(* ===== OUTER 10 ===== *)
GVL_test.stCase.aOuters[10].sOuterCode    := 'OUTER10';
GVL_test.stCase.aOuters[10].nOutersStatus := 5;
// packs 1..10
GVL_test.stCase.aOuters[10].aPacks[1].sPackCode   := 'PACK01OUTER10';
GVL_test.stCase.aOuters[10].aPacks[1].nPackStatus := 5;
GVL_test.stCase.aOuters[10].aPacks[2].sPackCode   := 'PACK02OUTER10';
GVL_test.stCase.aOuters[10].aPacks[2].nPackStatus := 5;
GVL_test.stCase.aOuters[10].aPacks[3].sPackCode   := 'PACK03OUTER10';
GVL_test.stCase.aOuters[10].aPacks[3].nPackStatus := 5;
GVL_test.stCase.aOuters[10].aPacks[4].sPackCode   := 'PACK04OUTER10';
GVL_test.stCase.aOuters[10].aPacks[4].nPackStatus := 5;
GVL_test.stCase.aOuters[10].aPacks[5].sPackCode   := 'PACK05OUTER10';
GVL_test.stCase.aOuters[10].aPacks[5].nPackStatus := 5;
GVL_test.stCase.aOuters[10].aPacks[6].sPackCode   := 'PACK06OUTER10';
GVL_test.stCase.aOuters[10].aPacks[6].nPackStatus := 5;
GVL_test.stCase.aOuters[10].aPacks[7].sPackCode   := 'PACK07OUTER10';
GVL_test.stCase.aOuters[10].aPacks[7].nPackStatus := 5;
GVL_test.stCase.aOuters[10].aPacks[8].sPackCode   := 'PACK08OUTER10';
GVL_test.stCase.aOuters[10].aPacks[8].nPackStatus := 5;
GVL_test.stCase.aOuters[10].aPacks[9].sPackCode   := 'PACK09OUTER10';
GVL_test.stCase.aOuters[10].aPacks[9].nPackStatus := 5;
GVL_test.stCase.aOuters[10].aPacks[10].sPackCode  := 'PACK10OUTER10';
GVL_test.stCase.aOuters[10].aPacks[10].nPackStatus := 5;
////////////////////////////////////////////////////////////////////////////////////
(* ===== OUTER 11 ===== *)
GVL_test.stCase.aOuters[11].sOuterCode    := 'OUTER1';
GVL_test.stCase.aOuters[11].nOutersStatus := 5;
// packs 1..10
GVL_test.stCase.aOuters[11].aPacks[1].sPackCode   := 'PACK01OUTER11';
GVL_test.stCase.aOuters[11].aPacks[1].nPackStatus := 5;
GVL_test.stCase.aOuters[11].aPacks[2].sPackCode   := 'PACK02OUTER11';
GVL_test.stCase.aOuters[11].aPacks[2].nPackStatus := 5;
GVL_test.stCase.aOuters[11].aPacks[3].sPackCode   := 'PACK03OUTER11';
GVL_test.stCase.aOuters[11].aPacks[3].nPackStatus := 5;
GVL_test.stCase.aOuters[11].aPacks[4].sPackCode   := 'PACK04OUTER11';
GVL_test.stCase.aOuters[11].aPacks[4].nPackStatus := 5;
GVL_test.stCase.aOuters[11].aPacks[5].sPackCode   := 'PACK05OUTER11';
GVL_test.stCase.aOuters[11].aPacks[5].nPackStatus := 5;
GVL_test.stCase.aOuters[11].aPacks[6].sPackCode   := 'PACK06OUTER11';
GVL_test.stCase.aOuters[11].aPacks[6].nPackStatus := 5;
GVL_test.stCase.aOuters[11].aPacks[7].sPackCode   := 'PACK07OUTER11';
GVL_test.stCase.aOuters[11].aPacks[7].nPackStatus := 5;
GVL_test.stCase.aOuters[11].aPacks[8].sPackCode   := 'PACK08OUTER11';
GVL_test.stCase.aOuters[11].aPacks[8].nPackStatus := 5;
GVL_test.stCase.aOuters[11].aPacks[9].sPackCode   := 'PACK09OUTER11';
GVL_test.stCase.aOuters[11].aPacks[9].nPackStatus := 5;
GVL_test.stCase.aOuters[11].aPacks[10].sPackCode  := 'PACK10OUTER11';
GVL_test.stCase.aOuters[11].aPacks[10].nPackStatus := 5;

(* ===== OUTER 12 ===== *)
GVL_test.stCase.aOuters[12].sOuterCode    := 'OUTER2';
GVL_test.stCase.aOuters[12].nOutersStatus := 5;
// packs 1..10
GVL_test.stCase.aOuters[12].aPacks[1].sPackCode   := 'PACK01OUTER12';
GVL_test.stCase.aOuters[12].aPacks[1].nPackStatus := 5;
GVL_test.stCase.aOuters[12].aPacks[2].sPackCode   := 'PACK02OUTER12';
GVL_test.stCase.aOuters[12].aPacks[2].nPackStatus := 5;
GVL_test.stCase.aOuters[12].aPacks[3].sPackCode   := 'PACK03OUTER12';
GVL_test.stCase.aOuters[12].aPacks[3].nPackStatus := 5;
GVL_test.stCase.aOuters[12].aPacks[4].sPackCode   := 'PACK04OUTER12';
GVL_test.stCase.aOuters[12].aPacks[4].nPackStatus := 5;
GVL_test.stCase.aOuters[12].aPacks[5].sPackCode   := 'PACK05OUTER12';
GVL_test.stCase.aOuters[12].aPacks[5].nPackStatus := 5;
GVL_test.stCase.aOuters[12].aPacks[6].sPackCode   := 'PACK06OUTER12';
GVL_test.stCase.aOuters[12].aPacks[6].nPackStatus := 5;
GVL_test.stCase.aOuters[12].aPacks[7].sPackCode   := 'PACK07OUTER12';
GVL_test.stCase.aOuters[12].aPacks[7].nPackStatus := 5;
GVL_test.stCase.aOuters[12].aPacks[8].sPackCode   := 'PACK08OUTER12';
GVL_test.stCase.aOuters[12].aPacks[8].nPackStatus := 5;
GVL_test.stCase.aOuters[12].aPacks[9].sPackCode   := 'PACK09OUTER12';
GVL_test.stCase.aOuters[12].aPacks[9].nPackStatus := 5;
GVL_test.stCase.aOuters[12].aPacks[10].sPackCode  := 'PACK10OUTER12';
GVL_test.stCase.aOuters[12].aPacks[10].nPackStatus := 5;

(* ===== OUTER 3 ===== *)
GVL_test.stCase.aOuters[3].sOuterCode    := 'OUTER3';
GVL_test.stCase.aOuters[3].nOutersStatus := 5;
// packs 1..10
GVL_test.stCase.aOuters[3].aPacks[1].sPackCode   := 'PACK01OUTER3';
GVL_test.stCase.aOuters[3].aPacks[1].nPackStatus := 5;
GVL_test.stCase.aOuters[3].aPacks[2].sPackCode   := 'PACK02OUTER3';
GVL_test.stCase.aOuters[3].aPacks[2].nPackStatus := 5;
GVL_test.stCase.aOuters[3].aPacks[3].sPackCode   := 'PACK03OUTER3';
GVL_test.stCase.aOuters[3].aPacks[3].nPackStatus := 5;
GVL_test.stCase.aOuters[3].aPacks[4].sPackCode   := 'PACK04OUTER3';
GVL_test.stCase.aOuters[3].aPacks[4].nPackStatus := 5;
GVL_test.stCase.aOuters[3].aPacks[5].sPackCode   := 'PACK05OUTER3';
GVL_test.stCase.aOuters[3].aPacks[5].nPackStatus := 5;
GVL_test.stCase.aOuters[3].aPacks[6].sPackCode   := 'PACK06OUTER3';
GVL_test.stCase.aOuters[3].aPacks[6].nPackStatus := 5;
GVL_test.stCase.aOuters[3].aPacks[7].sPackCode   := 'PACK07OUTER3';
GVL_test.stCase.aOuters[3].aPacks[7].nPackStatus := 5;
GVL_test.stCase.aOuters[3].aPacks[8].sPackCode   := 'PACK08OUTER3';
GVL_test.stCase.aOuters[3].aPacks[8].nPackStatus := 5;
GVL_test.stCase.aOuters[3].aPacks[9].sPackCode   := 'PACK09OUTER3';
GVL_test.stCase.aOuters[3].aPacks[9].nPackStatus := 5;
GVL_test.stCase.aOuters[3].aPacks[10].sPackCode  := 'PACK10OUTER3';
GVL_test.stCase.aOuters[3].aPacks[10].nPackStatus := 5;

(* ===== OUTER 4 ===== *)
GVL_test.stCase.aOuters[4].sOuterCode    := 'OUTER4';
GVL_test.stCase.aOuters[4].nOutersStatus := 5;
// packs 1..10
GVL_test.stCase.aOuters[4].aPacks[1].sPackCode   := 'PACK01OUTER4';
GVL_test.stCase.aOuters[4].aPacks[1].nPackStatus := 5;
GVL_test.stCase.aOuters[4].aPacks[2].sPackCode   := 'PACK02OUTER4';
GVL_test.stCase.aOuters[4].aPacks[2].nPackStatus := 5;
GVL_test.stCase.aOuters[4].aPacks[3].sPackCode   := 'PACK03OUTER4';
GVL_test.stCase.aOuters[4].aPacks[3].nPackStatus := 5;
GVL_test.stCase.aOuters[4].aPacks[4].sPackCode   := 'PACK04OUTER4';
GVL_test.stCase.aOuters[4].aPacks[4].nPackStatus := 5;
GVL_test.stCase.aOuters[4].aPacks[5].sPackCode   := 'PACK05OUTER4';
GVL_test.stCase.aOuters[4].aPacks[5].nPackStatus := 5;
GVL_test.stCase.aOuters[4].aPacks[6].sPackCode   := 'PACK06OUTER4';
GVL_test.stCase.aOuters[4].aPacks[6].nPackStatus := 5;
GVL_test.stCase.aOuters[4].aPacks[7].sPackCode   := 'PACK07OUTER4';
GVL_test.stCase.aOuters[4].aPacks[7].nPackStatus := 5;
GVL_test.stCase.aOuters[4].aPacks[8].sPackCode   := 'PACK08OUTER4';
GVL_test.stCase.aOuters[4].aPacks[8].nPackStatus := 5;
GVL_test.stCase.aOuters[4].aPacks[9].sPackCode   := 'PACK09OUTER4';
GVL_test.stCase.aOuters[4].aPacks[9].nPackStatus := 5;
GVL_test.stCase.aOuters[4].aPacks[10].sPackCode  := 'PACK10OUTER4';
GVL_test.stCase.aOuters[4].aPacks[10].nPackStatus := 5;

(* ===== OUTER 5 ===== *)
GVL_test.stCase.aOuters[5].sOuterCode    := 'OUTER5';
GVL_test.stCase.aOuters[5].nOutersStatus := 5;
// packs 1..10
GVL_test.stCase.aOuters[5].aPacks[1].sPackCode   := 'PACK01OUTER5';
GVL_test.stCase.aOuters[5].aPacks[1].nPackStatus := 5;
GVL_test.stCase.aOuters[5].aPacks[2].sPackCode   := 'PACK02OUTER5';
GVL_test.stCase.aOuters[5].aPacks[2].nPackStatus := 5;
GVL_test.stCase.aOuters[5].aPacks[3].sPackCode   := 'PACK03OUTER5';
GVL_test.stCase.aOuters[5].aPacks[3].nPackStatus := 5;
GVL_test.stCase.aOuters[5].aPacks[4].sPackCode   := 'PACK04OUTER5';
GVL_test.stCase.aOuters[5].aPacks[4].nPackStatus := 5;
GVL_test.stCase.aOuters[5].aPacks[5].sPackCode   := 'PACK05OUTER5';
GVL_test.stCase.aOuters[5].aPacks[5].nPackStatus := 5;
GVL_test.stCase.aOuters[5].aPacks[6].sPackCode   := 'PACK06OUTER5';
GVL_test.stCase.aOuters[5].aPacks[6].nPackStatus := 5;
GVL_test.stCase.aOuters[5].aPacks[7].sPackCode   := 'PACK07OUTER5';
GVL_test.stCase.aOuters[5].aPacks[7].nPackStatus := 5;
GVL_test.stCase.aOuters[5].aPacks[8].sPackCode   := 'PACK08OUTER5';
GVL_test.stCase.aOuters[5].aPacks[8].nPackStatus := 5;
GVL_test.stCase.aOuters[5].aPacks[9].sPackCode   := 'PACK09OUTER5';
GVL_test.stCase.aOuters[5].aPacks[9].nPackStatus := 5;
GVL_test.stCase.aOuters[5].aPacks[10].sPackCode  := 'PACK10OUTER5';
GVL_test.stCase.aOuters[5].aPacks[10].nPackStatus := 5;

(* ===== OUTER 6 ===== *)
GVL_test.stCase.aOuters[6].sOuterCode    := 'OUTER6';
GVL_test.stCase.aOuters[6].nOutersStatus := 5;
// packs 1..10
GVL_test.stCase.aOuters[6].aPacks[1].sPackCode   := 'PACK01OUTER6';
GVL_test.stCase.aOuters[6].aPacks[1].nPackStatus := 5;
GVL_test.stCase.aOuters[6].aPacks[2].sPackCode   := 'PACK02OUTER6';
GVL_test.stCase.aOuters[6].aPacks[2].nPackStatus := 5;
GVL_test.stCase.aOuters[6].aPacks[3].sPackCode   := 'PACK03OUTER6';
GVL_test.stCase.aOuters[6].aPacks[3].nPackStatus := 5;
GVL_test.stCase.aOuters[6].aPacks[4].sPackCode   := 'PACK04OUTER6';
GVL_test.stCase.aOuters[6].aPacks[4].nPackStatus := 5;
GVL_test.stCase.aOuters[6].aPacks[5].sPackCode   := 'PACK05OUTER6';
GVL_test.stCase.aOuters[6].aPacks[5].nPackStatus := 5;
GVL_test.stCase.aOuters[6].aPacks[6].sPackCode   := 'PACK06OUTER6';
GVL_test.stCase.aOuters[6].aPacks[6].nPackStatus := 5;
GVL_test.stCase.aOuters[6].aPacks[7].sPackCode   := 'PACK07OUTER6';
GVL_test.stCase.aOuters[6].aPacks[7].nPackStatus := 5;
GVL_test.stCase.aOuters[6].aPacks[8].sPackCode   := 'PACK08OUTER6';
GVL_test.stCase.aOuters[6].aPacks[8].nPackStatus := 5;
GVL_test.stCase.aOuters[6].aPacks[9].sPackCode   := 'PACK09OUTER6';
GVL_test.stCase.aOuters[6].aPacks[9].nPackStatus := 5;
GVL_test.stCase.aOuters[6].aPacks[10].sPackCode  := 'PACK10OUTER6';
GVL_test.stCase.aOuters[6].aPacks[10].nPackStatus := 5;

(* ===== OUTER 7 ===== *)
GVL_test.stCase.aOuters[7].sOuterCode    := 'OUTER7';
GVL_test.stCase.aOuters[7].nOutersStatus := 5;
// packs 1..10
GVL_test.stCase.aOuters[7].aPacks[1].sPackCode   := 'PACK01OUTER7';
GVL_test.stCase.aOuters[7].aPacks[1].nPackStatus := 5;
GVL_test.stCase.aOuters[7].aPacks[2].sPackCode   := 'PACK02OUTER7';
GVL_test.stCase.aOuters[7].aPacks[2].nPackStatus := 5;
GVL_test.stCase.aOuters[7].aPacks[3].sPackCode   := 'PACK03OUTER7';
GVL_test.stCase.aOuters[7].aPacks[3].nPackStatus := 5;
GVL_test.stCase.aOuters[7].aPacks[4].sPackCode   := 'PACK04OUTER7';
GVL_test.stCase.aOuters[7].aPacks[4].nPackStatus := 5;
GVL_test.stCase.aOuters[7].aPacks[5].sPackCode   := 'PACK05OUTER7';
GVL_test.stCase.aOuters[7].aPacks[5].nPackStatus := 5;
GVL_test.stCase.aOuters[7].aPacks[6].sPackCode   := 'PACK06OUTER7';
GVL_test.stCase.aOuters[7].aPacks[6].nPackStatus := 5;
GVL_test.stCase.aOuters[7].aPacks[7].sPackCode   := 'PACK07OUTER7';
GVL_test.stCase.aOuters[7].aPacks[7].nPackStatus := 5;
GVL_test.stCase.aOuters[7].aPacks[8].sPackCode   := 'PACK08OUTER7';
GVL_test.stCase.aOuters[7].aPacks[8].nPackStatus := 5;
GVL_test.stCase.aOuters[7].aPacks[9].sPackCode   := 'PACK09OUTER7';
GVL_test.stCase.aOuters[7].aPacks[9].nPackStatus := 5;
GVL_test.stCase.aOuters[7].aPacks[10].sPackCode  := 'PACK10OUTER7';
GVL_test.stCase.aOuters[7].aPacks[10].nPackStatus := 5;

(* ===== OUTER 8 ===== *)
GVL_test.stCase.aOuters[8].sOuterCode    := 'OUTER8';
GVL_test.stCase.aOuters[8].nOutersStatus := 5;
// packs 1..10
GVL_test.stCase.aOuters[8].aPacks[1].sPackCode   := 'PACK01OUTER8';
GVL_test.stCase.aOuters[8].aPacks[1].nPackStatus := 5;
GVL_test.stCase.aOuters[8].aPacks[2].sPackCode   := 'PACK02OUTER8';
GVL_test.stCase.aOuters[8].aPacks[2].nPackStatus := 5;
GVL_test.stCase.aOuters[8].aPacks[3].sPackCode   := 'PACK03OUTER8';
GVL_test.stCase.aOuters[8].aPacks[3].nPackStatus := 5;
GVL_test.stCase.aOuters[8].aPacks[4].sPackCode   := 'PACK04OUTER8';
GVL_test.stCase.aOuters[8].aPacks[4].nPackStatus := 5;
GVL_test.stCase.aOuters[8].aPacks[5].sPackCode   := 'PACK05OUTER8';
GVL_test.stCase.aOuters[8].aPacks[5].nPackStatus := 5;
GVL_test.stCase.aOuters[8].aPacks[6].sPackCode   := 'PACK06OUTER8';
GVL_test.stCase.aOuters[8].aPacks[6].nPackStatus := 5;
GVL_test.stCase.aOuters[8].aPacks[7].sPackCode   := 'PACK07OUTER8';
GVL_test.stCase.aOuters[8].aPacks[7].nPackStatus := 5;
GVL_test.stCase.aOuters[8].aPacks[8].sPackCode   := 'PACK08OUTER8';
GVL_test.stCase.aOuters[8].aPacks[8].nPackStatus := 5;
GVL_test.stCase.aOuters[8].aPacks[9].sPackCode   := 'PACK09OUTER8';
GVL_test.stCase.aOuters[8].aPacks[9].nPackStatus := 5;
GVL_test.stCase.aOuters[8].aPacks[10].sPackCode  := 'PACK10OUTER8';
GVL_test.stCase.aOuters[8].aPacks[10].nPackStatus := 5;

(* ===== OUTER 9 ===== *)
GVL_test.stCase.aOuters[9].sOuterCode    := 'OUTER9';
GVL_test.stCase.aOuters[9].nOutersStatus := 5;
// packs 1..10
GVL_test.stCase.aOuters[9].aPacks[1].sPackCode   := 'PACK01OUTER9';
GVL_test.stCase.aOuters[9].aPacks[1].nPackStatus := 5;
GVL_test.stCase.aOuters[9].aPacks[2].sPackCode   := 'PACK02OUTER9';
GVL_test.stCase.aOuters[9].aPacks[2].nPackStatus := 5;
GVL_test.stCase.aOuters[9].aPacks[3].sPackCode   := 'PACK03OUTER9';
GVL_test.stCase.aOuters[9].aPacks[3].nPackStatus := 5;
GVL_test.stCase.aOuters[9].aPacks[4].sPackCode   := 'PACK04OUTER9';
GVL_test.stCase.aOuters[9].aPacks[4].nPackStatus := 5;
GVL_test.stCase.aOuters[9].aPacks[5].sPackCode   := 'PACK05OUTER9';
GVL_test.stCase.aOuters[9].aPacks[5].nPackStatus := 5;
GVL_test.stCase.aOuters[9].aPacks[6].sPackCode   := 'PACK06OUTER9';
GVL_test.stCase.aOuters[9].aPacks[6].nPackStatus := 5;
GVL_test.stCase.aOuters[9].aPacks[7].sPackCode   := 'PACK07OUTER9';
GVL_test.stCase.aOuters[9].aPacks[7].nPackStatus := 5;
GVL_test.stCase.aOuters[9].aPacks[8].sPackCode   := 'PACK08OUTER9';
GVL_test.stCase.aOuters[9].aPacks[8].nPackStatus := 5;
GVL_test.stCase.aOuters[9].aPacks[9].sPackCode   := 'PACK09OUTER9';
GVL_test.stCase.aOuters[9].aPacks[9].nPackStatus := 5;
GVL_test.stCase.aOuters[9].aPacks[10].sPackCode  := 'PACK10OUTER9';
GVL_test.stCase.aOuters[9].aPacks[10].nPackStatus := 5;

(* ===== OUTER 10 ===== *)
GVL_test.stCase.aOuters[10].sOuterCode    := 'OUTER10';
GVL_test.stCase.aOuters[10].nOutersStatus := 5;
// packs 1..10
GVL_test.stCase.aOuters[10].aPacks[1].sPackCode   := 'PACK01OUTER10';
GVL_test.stCase.aOuters[10].aPacks[1].nPackStatus := 5;
GVL_test.stCase.aOuters[10].aPacks[2].sPackCode   := 'PACK02OUTER10';
GVL_test.stCase.aOuters[10].aPacks[2].nPackStatus := 5;
GVL_test.stCase.aOuters[10].aPacks[3].sPackCode   := 'PACK03OUTER10';
GVL_test.stCase.aOuters[10].aPacks[3].nPackStatus := 5;
GVL_test.stCase.aOuters[10].aPacks[4].sPackCode   := 'PACK04OUTER10';
GVL_test.stCase.aOuters[10].aPacks[4].nPackStatus := 5;
GVL_test.stCase.aOuters[10].aPacks[5].sPackCode   := 'PACK05OUTER10';
GVL_test.stCase.aOuters[10].aPacks[5].nPackStatus := 5;
GVL_test.stCase.aOuters[10].aPacks[6].sPackCode   := 'PACK06OUTER10';
GVL_test.stCase.aOuters[10].aPacks[6].nPackStatus := 5;
GVL_test.stCase.aOuters[10].aPacks[7].sPackCode   := 'PACK07OUTER10';
GVL_test.stCase.aOuters[10].aPacks[7].nPackStatus := 5;
GVL_test.stCase.aOuters[10].aPacks[8].sPackCode   := 'PACK08OUTER10';
GVL_test.stCase.aOuters[10].aPacks[8].nPackStatus := 5;
GVL_test.stCase.aOuters[10].aPacks[9].sPackCode   := 'PACK09OUTER10';
GVL_test.stCase.aOuters[10].aPacks[9].nPackStatus := 5;
GVL_test.stCase.aOuters[10].aPacks[10].sPackCode  := 'PACK10OUTER10';
GVL_test.stCase.aOuters[10].aPacks[10].nPackStatus := 5;
END_ACTION

ACTION CaseDataAdd:
(*     outer 1 data     *)
GVL_test.stCase.aOuters[1].sOuterCode 	:= 'OUTER1';
GVL_test.stCase.aOuters[1].nOutersStatus	:= 5;
// packs 1..10
GVL_test.stCase.aOuters[1].aPacks[1].sPackCode 		:= 'PACK01OUTER1';
GVL_test.stCase.aOuters[1].aPacks[1].nPackStatus 	:= 5;
GVL_test.stCase.aOuters[1].aPacks[2].sPackCode 		:= 'PACK02OUTER1';
GVL_test.stCase.aOuters[1].aPacks[2].nPackStatus 	:= 5;
GVL_test.stCase.aOuters[1].aPacks[3].sPackCode 		:= 'PACK03OUTER1';
GVL_test.stCase.aOuters[1].aPacks[3].nPackStatus 	:= 5;
GVL_test.stCase.aOuters[1].aPacks[4].sPackCode 		:= 'PACK04OUTER1';
GVL_test.stCase.aOuters[1].aPacks[4].nPackStatus 	:= 5;
GVL_test.stCase.aOuters[1].aPacks[5].sPackCode 		:= 'PACK05OUTER1';
GVL_test.stCase.aOuters[1].aPacks[5].nPackStatus 	:= 5;
GVL_test.stCase.aOuters[1].aPacks[6].sPackCode 		:= 'PACK06OUTER1';
GVL_test.stCase.aOuters[1].aPacks[6].nPackStatus 	:= 5;
GVL_test.stCase.aOuters[1].aPacks[7].sPackCode 		:= 'PACK07OUTER1';
GVL_test.stCase.aOuters[1].aPacks[7].nPackStatus 	:= 5;
GVL_test.stCase.aOuters[1].aPacks[8].sPackCode 		:= 'PACK08OUTER1';
GVL_test.stCase.aOuters[1].aPacks[8].nPackStatus 	:= 5;
GVL_test.stCase.aOuters[1].aPacks[9].sPackCode 		:= 'PACK09OUTER1';
GVL_test.stCase.aOuters[1].aPacks[9].nPackStatus 	:= 5;
GVL_test.stCase.aOuters[1].aPacks[10].sPackCode 	:= 'PACK10OUTER1';
GVL_test.stCase.aOuters[1].aPacks[10].nPackStatus 	:= 5;



(*     outer 1 data     *)
GVL_test.stCase.aOuters[2].sOuterCode 	:= 'OUTER1';
GVL_test.stCase.aOuters[2].nOutersStatus	:= 5;
// packs 1 data
GVL_test.stCase.aOuters[2].aPacks[1].sPackCode 	:= 'PACK01OUTER1';
GVL_test.stCase.aOuters[2].aPacks[1].nPackStatus := 5;
// packs 2 data
GVL_test.stCase.aOuters[2].aPacks[2].sPackCode 	:= 'PACK02OUTER1';
GVL_test.stCase.aOuters[2].aPacks[2].nPackStatus := 5;
// packs 3 data
GVL_test.stCase.aOuters[2].aPacks[3].sPackCode 	:= 'PACK03OUTER1';
GVL_test.stCase.aOuters[2].aPacks[3].nPackStatus := 5;

(*     outer 2 data     *)
GVL_test.stCase.aOuters[2].sOuterCode 	:= 'OUTER2';
GVL_test.stCase.aOuters[2].nOutersStatus	:= 5;
// packs 1 data
GVL_test.stCase.aOuters[2].aPacks[1].sPackCode 	:= 'PACK01OUTER2';
GVL_test.stCase.aOuters[2].aPacks[1].nPackStatus := 5;
// packs 2 data
GVL_test.stCase.aOuters[2].aPacks[2].sPackCode 	:= 'PACK02OUTER2';
GVL_test.stCase.aOuters[2].aPacks[2].nPackStatus := 5;
// packs 3 data
GVL_test.stCase.aOuters[2].aPacks[3].sPackCode 	:= 'PACK03OUTER2';
GVL_test.stCase.aOuters[2].aPacks[3].nPackStatus := 5;


(*     outer 3 data     *)
GVL_test.stCase.aOuters[3].sOuterCode 	:= 'OUTER3';
GVL_test.stCase.aOuters[3].nOutersStatus	:= 5;
// packs 1 data
GVL_test.stCase.aOuters[3].aPacks[1].sPackCode 	:= 'PACK01OUTER3';
GVL_test.stCase.aOuters[3].aPacks[1].nPackStatus := 5;
// packs 2 data
GVL_test.stCase.aOuters[3].aPacks[2].sPackCode 	:= 'PACK02OUTER3';
GVL_test.stCase.aOuters[3].aPacks[2].nPackStatus := 5;
// packs 3 data
GVL_test.stCase.aOuters[3].aPacks[3].sPackCode 	:= 'PACK03OUTER3';
GVL_test.stCase.aOuters[3].aPacks[3].nPackStatus := 5;
END_ACTION

ACTION FullFilOuter:

rTrigDataFill(CLK := bDataFill);

IF rTrigDataFill.Q THEN
	
	FOR iOuter := 1 TO 50 DO
		(* Ustaw outer *)
		GVL_test.stCaseFull.aOuters[iOuter].sOuterCode    := CONCAT('OUTER', INT_TO_STRING(iOuter));
		GVL_test.stCaseFull.aOuters[iOuter].nOutersStatus := 5;
		
		FOR iPack := 1 TO 10 DO
			(* Pack number z zerami *)
			sPackNum := CONCAT('0', INT_TO_STRING(iPack));  (* dla 1-9: '01'-'09' *)
			IF iPack = 10 THEN
				sPackNum := '10';
			END_IF;
			
			(* Outer number z zerami dla 1-9 *)
			sOuterNum := CONCAT('0', INT_TO_STRING(iOuter));
			IF iOuter >= 10 THEN
				sOuterNum := INT_TO_STRING(iOuter);
			END_IF;
			
			(* Sklej pack code *)
			sPackCode := CONCAT(CONCAT('PACK', sPackNum), CONCAT('OUTER', sOuterNum));
			
			(* Przypisz *)
			GVL_test.stCaseFull.aOuters[iOuter].aPacks[iPack].sPackCode   := sPackCode;
			GVL_test.stCaseFull.aOuters[iOuter].aPacks[iPack].nPackStatus := 5;
		END_FOR;
	END_FOR;
	
END_IF
END_ACTION

END_PROGRAM

// ---- POUs/_Utilites/Tests/PRG_TestCamera.TcPOU
PROGRAM PRG_TestCamera
VAR
	nMaxBytes: UDINT;
	strTCPRxString: STRING(255);
	
	strTargetIPAddr		: T_IPv4Addr := '192.168.1.44';	
	arrTargetIPAddr		: T_IPv4AddrArr;
	nSyncOffset			: DINT;		
	nSyncOffset_1		: DINT;	
	tTaskTime			: TIME := T#200MS;
	sString_1			: STRING(255);
	sString_2			: STRING(255);
	sConcuted			: STRING(1023);
	bConcuted			: BOOL;
	
	nSize_1				: UINT;
	nSize_2				: UINT;
	nSize_3				: UDINT;
	nStatusByte			: BYTE;
	bitNO				: USINT := 6;
	nBytesQuantity		: INT :=1;
	nBytePosition		: INT :=5;
	sString_4			: STRING(255);
	strTCPRxDebug		: ARRAY[1..20] OF  STRING(100);
	nSizeTCPRxDebug		: UINT;
	sStringTest			: STRING(100) := '_STRING_W_PIERWSZEJ_TABLICY_';
	nIndex				: INT;
	nSizeTCPRxDebug_1	: UINT;
END_VAR


nMaxBytes := SIZEOF(strTCPRxString) - INT_TO_UDINT(LEN(strTCPRxString) - 1);

arrTargetIPAddr := F_ScanIPv4AddrIds(strTargetIPAddr);
nSyncOffset := arrTargetIPAddr[3] MOD 10;

nSyncOffset_1		:= nSyncOffset * TIME_TO_DINT(tTaskTime);

sString_1 := '_1st_RGST$07$04;$02CT=11;DS=HTTPS://Y2WM.CN/99.1000.1/AC12bTPL1003RC78N3TRBUQME1J4XR9ZC;OG=0;QS=1;UE=1.00;XP=19;YP=-5;AP=91;CS=05.6;SC=0056;PN=1;$03$04';
sString_2 := '_2nd_RGST$07$04;$02CT=11;DS=HTTPS://Y2WM.CN/99.1000.1/AC12bTPL1003RC78N3TRBUQME1J4XR9ZC;OG=0;QS=1;UE=1.00;XP=19;YP=-5;AP=91;CS=05.6;SC=0056;PN=1;$03$04';

bConcuted := CONCAT2(pSrcString1 := ADR(sString_1), pSrcString2 := ADR(sString_2), pDstString := ADR(sConcuted), SIZEOF(sConcuted));

nSize_1 := LEN(sString_1);
nSize_2 := LEN(sString_2);
nSize_3 := LEN2(ADR(sConcuted));

nStatusByte := ASC(MID(sString_1, nBytesQuantity, bitNO));
nStatusByte.0;
nStatusByte.1;
nStatusByte.2;
nStatusByte.3;
nStatusByte.4;
nStatusByte.5;
nStatusByte.6;
nStatusByte.7;

sString_4	:= MID(sString_1, 4, 6);

//strTCPRxDebug[1] := sStringTest;

FOR nIndex := 1 TO 20 DO
	strTCPRxDebug[nIndex] := CONCAT(CONCAT('_MESSAGE_NO_', INT_TO_STRING(nIndex)), '_'); 	
END_FOR

nSizeTCPRxDebug 	:= SIZEOF(strTCPRxDebug);
nSizeTCPRxDebug_1	:= SIZEOF(strTCPRxDebug[1]);

MEMMOVE(ADR(strTCPRxDebug[2]), ADR(strTCPRxDebug[1]), SIZEOF(strTCPRxDebug)-SIZEOF(strTCPRxDebug[1]));

END_PROGRAM
